// TIA Portal V18 export
// export: Created 2025-12-01T12:38:44.2125882Z, ExportSetting None, DisplayName Totally Integrated Automation Portal, DisplayVersion V18 Update 5, DisplayName TIA Portal Openness, DisplayVersion V18 Update 5, DisplayName TIA Portal Teamcenter Gateway, DisplayVersion V18, DisplayName TIA Portal Version Control Interface, DisplayVersion V18, DisplayName STEP 7 Professional, DisplayVersion V18 Update 5, DisplayName STEP 7 Safety, DisplayVersion V18, DisplayName WinCC Professional, DisplayVersion V18 Update 5
DATA_BLOCK "V90Servo_DB"   // DB2500
// stored: AutoNumber false, InstanceOfName V90_Servo, InstanceOfType FB
"V90_Servo"
   // VAR
   //    Servo_380A1 { S7_SetPoint := 'True'} : "fbV90Ctrl";
   //    Servo_381A1 { S7_SetPoint := 'True'} : "fbV90Ctrl";
   //    Servo_382A1 { S7_SetPoint := 'True'} : "fbV90Ctrl";
   //    Servo_383A1 { S7_SetPoint := 'True'} : "fbV90Ctrl";
   //    Servo1 { S7_SetPoint := 'True'} : "SevroStart&PosCheck";
   //    Servo2 { S7_SetPoint := 'True'} : "SevroStart&PosCheck";
   //    Servo3 { S7_SetPoint := 'True'} : "SevroStart&PosCheck";
   //    Servo4 { S7_SetPoint := 'True'} : "SevroStart&PosCheck";
   //    Servo2SafetyPos { S7_SetPoint := 'True'} : DInt;
   //    Servo4SafetyPos { S7_SetPoint := 'True'} : DInt;
   //    IEC_Timer_0_Instance { S7_SetPoint := 'True'} : TON_TIME;
   //    P { S7_SetPoint := 'True'} : Array[0..10] of Bool;
   // END_VAR
BEGIN
END_DATA_BLOCK
